FUNCTION Convert_LREAL_TO_DT : Hresult
VAR_INPUT
	in : LREAL;
	out : REFERENCE TO DT;
END_VAR
VAR
	converted : DT;
END_VAR
VAR CONSTANT
	INCOMPATIBLE : HRESULT := 16#9811070E;
END_VAR

converted := LREAL_TO_DT(in);

IF (DT_TO_LREAL(converted) <> in) THEN
	Convert_LREAL_TO_DT := INCOMPATIBLE;
	RETURN;
END_IF

out := converted;

END_FUNCTION

(* stored: Version 1.1.0.1, ProductVersion 3.1.4024.12
   POU Convert_LREAL_TO_DT: Id {c1752dac-1cdb-4989-b73f-bbb4a24e9736}, SpecialFunc None *)
